TYPE JSON_DriveList : ARRAY[0..39] OF JSON_Drive; END_TYPE

(* stored: Version 1.1.0.1
   DUT JSON_DriveList: Id {8bad7b7e-16dc-0d8a-03dd-b5bccc29e31c} *)
